Fanuc KAREL source: kf00116.KL

PROGRAM KF00116
%STACKSIZE=65535
%PRIORITY=65535
%NOLOCKGROUP
VAR
I : INTEGER
J : INTEGER
X : REAL
Y : REAL
B : BOOLEAN
C : BOOLEAN
TXT : STRING[80]
TXT2 : STRING[80]
AI : ARRAY[4] OF INTEGER
BI : ARRAY[4] OF INTEGER
P : XYZWPR
JP : JOINTPOS9
PF : POSITION
STATUS : INTEGER
-- UNRESOLVED DECLARATIONS (source type spelling not recovered)
-- V1 : TYPE_0x0013 (type_u16=0x0013)
-- V2 : TYPE_0x0013 (type_u16=0x0013)
ROUTINE FACT(P1 : INTEGER) : INTEGER FROM KF00116
ROUTINE FACT
BEGIN
IF (P1 <=1) THEN
RETURN(1)
ELSE
-- UNSAFE_SOURCE_IR line 25: CALL_RESULT FACT(ARG_1_UNRESOLVED)
ENDIF
-- UNRESOLVED_PC line 27 opcodes [7F] marker_code=73
END FACT
BEGIN
I=FACT(3)
END KF00116
